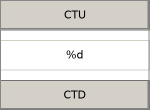
VISUALIZATION FP_Counter  // 150x110
VAR_IN_OUT
	o_CTU		: BOOL;
	o_CTD		: BOOL;
END_VAR

VAR_INPUT
	ctnValue	: INT;
END_VAR
    Group (0,0 150x110)
        Button (0,0 150x30), "CTU"
            tap btnCTU
        Button (0,80 150x30), "CTD"
            tap btuCTD
        Textfield (0,40 150x30), "%d", text variable: ctnValue
END_VISUALIZATION

(* stored: Version 1.1.0.1, ProductVersion 3.1.4024.12
   Visu FP_Counter: Id {6429dbe3-3649-4f3d-9bb9-fe8c7b6a95ab} *)
